Universal Robots PolyScope program: Pick and drop.urp

Program Pick and drop (createdIn=3.2.18654 lastSavedIn=3.2.18654 directory=/home/ur/ursim-3.2/programs installation=default robotSerialNumber=2014359999)
Calibrated DH parameters: a=[0, -0.425, -0.39225, 0, 0, 0]; d=[0.089159, 0, 0, 0.10915, 0.09465, 0.0823]; alpha=[1.570796, 0, 0, 1.570796, -1.570796, 0]; deltaTheta=[0, 0, 0, 0, 0, 0]
Robot Program (runOnlyOnce=false motionType=MoveJ speed=1.047198 acceleration=1.396263 recalculateMotions=false)
  MoveJ speed 60 deg/s, acceleration 80 deg/s^2 (recalculateMotions=false)
    Waypoint Home: 
  MoveJ speed 60 deg/s, acceleration 80 deg/s^2 (recalculateMotions=true)
    Waypoint Pre_pick: 
  MoveL speed 250 mm/s, acceleration 1200 mm/s^2 (recalculateMotions=false) feature=Base
    Waypoint Pick: 
